TYPE ST_HMI_InputSourceCtrl : 
STRUCT
	nActiveRecordIdx: INT;
	
	dtSelectedRangeStart: DCTIMESTRUCT;
	dtSelectedRangeEnd: DCTIMESTRUCT;
	
	bStart: BOOL;
	bCancel: BOOL;
	bPause: BOOL;
	bReset: BOOL;
END_STRUCT
END_TYPE

(* stored: DUT ST_HMI_InputSourceCtrl: Id 2a6e906b-8ab2-4237-a599-8cf3cbcc36d1 *)
